SUBAPPLICATION Uebung_012g_AR2 (* Numeric Value Input PHYS und Speichern INI via AR2 (bidirektional) - NumericValue_TO_AR2 direkt an ein INI_AR2 angeschlossen *)
  (* Standard: 61499-2; Description: Copyright (c) 2026 Meisterschulen am Ostbahnhof This program and the accompanying materials are made available under the terms of the Eclipse Public License 2.0 which is available at https://www.eclipse.org/legal/epl-2.0/ SPDX-License-Identifier: EPL-2.0 *)
  (* Version 1.0, 2026-04-24, Franz Höpfinger, Meisterschulen am Ostbahnhof, AR adapter variant of Uebung_012g, plain without subapp *)
  (* Version 2.0, 2026-08-31, Franz Höpfinger, Meisterschulen am Ostbahnhof, AR2 variant: MyLib::sys::NumericValue_TO_AR2 (VT-Eingabefeld gelesen, als AR2 weitergereicht, persistiert NICHT selbst) direkt an INI_AR2 (persistiert via AR2 Socket) angeschlossen - INI-Gegenstueck zu Uebung_012d_AR2 (NVS) *)
  PACKAGE Uebungen;
  IMPORT Uebungen::const::NVS::NVS_Keys::KEY_I1_STORE;
  IMPORT Uebungen::const::NVS::NVS_Keys::SECTION_I1_STORE;
  IMPORT Uebungen::const::UT::DefaultPool_Numeric::InputNumber_I3_N;
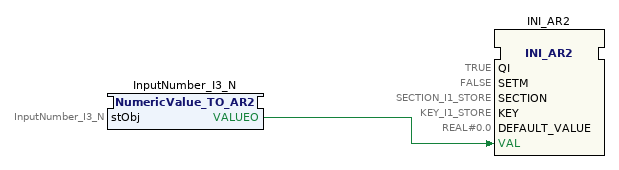
  (* NumericValue_TO_AR2 speichert NICHTS selbst - es liest nur das VT-Eingabefeld (InputNumber_I3_N) und reicht den Wert als AR2 (bidirektional) weiter. Die eigentliche Speicherung passiert ausschliesslich in INI_AR2 rechts daneben. *)
  (* SETM=FALSE hier: das betrifft NICHT den Boot-Wert - der laedt immer automatisch (INIT -> INITO -> GET -> GETO -> Echo an NumericValue_TO_AR2 -> Anzeige, unabhaengig von SETM). SETM gilt nur fuer eine LIVE-Aenderung waehrend des laufenden Betriebs: mit SETM=FALSE wird ein frisch eingegebener Wert zwar gespeichert, aber die Bestaetigung nicht sofort zurueckgemeldet - erst der naechste Neustart zeigt ihn wieder korrekt an. Wo der frische Wert noch IM SELBEN Lauf sofort weiterverwendet wird (z.B. AR_CALIBRATE_SQ_REF.ZERO/SPAN fuer CO/CS), braucht es SETM=TRUE. *)
  FBS
    INI_AR2 : eclipse4diac::storage::INI_AR2(QI := TRUE, SETM := FALSE, SECTION := SECTION_I1_STORE, KEY := KEY_I1_STORE, DEFAULT_VALUE := REAL#0.0);
  END_FBS
  SUBAPPS
    InputNumber_I3_N : MyLib::sys::NumericValue_TO_AR2(stObj := InputNumber_I3_N);
  END_SUBAPPS
  ADAPTER_CONNECTIONS
    InputNumber_I3_N.VALUEO TO INI_AR2.VAL;
  END_CONNECTIONS
END_SUBAPPLICATION
